# EPICS substitutions: modules/event/evrSupport/Db/ioc/IOC-IN20-LS15evr.substitutions
#==============================================================================
#
# Abs:  LCLS EVR IOC records for IN20 LS15
#
# Name: IOC-IN20-LS15evr.substitutions
#
#==============================================================================
#
file evrLSXX.db
{
pattern { DEVICE        }
	{ EVR:IN20:LS15 }
}
